PROGRAM LadderExample
VAR
	input: BOOL;
	output: BOOL;
	input2: BOOL;
END_VAR

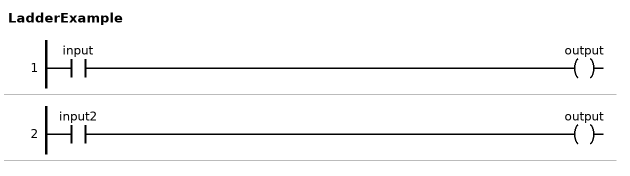
// NETWORK 1
output := input;

// NETWORK 2
output := input2;

END_PROGRAM

(* stored: Version 1.1.0.1, ProductVersion 3.1.4024.12
   POU LadderExample: Id {1b56824e-34e9-4b09-b43b-24d3e66681c3}, SpecialFunc None *)
